// TIA Portal V17 export
// export: Created 2022-06-27T13:58:59.0889884Z, ExportSetting WithDefaults, DisplayName Totally Integrated Automation Portal, DisplayVersion V17 Update 3, DisplayName TIA Portal Openness, DisplayVersion V17 Update 3, DisplayName TIA Portal Version Control Interface, DisplayVersion V17, DisplayName SINAMICS Startdrive Advanced, DisplayVersion V17 Update1, DisplayName SINAMICS Startdrive G110M, G120, G120C, G120D, G120P, G115D, DisplayVersion V17 Update1, DisplayName SINAMICS Startdrive G130, G150, S120, S150, SINAMICS MV, S210, DisplayVersion V17 Update1, DisplayName STEP 7 Professional, DisplayVersion V17 Update 3, DisplayName STEP 7 Safety, DisplayVersion V17, DisplayName WinCC UA Professional, DisplayVersion V17 Update 3
FUNCTION_BLOCK "S063_PROTECTION"   // FB63, LAD
{ S7_Optimized_Access := 'TRUE' }
VERSION : 0.1
// stored: AutoNumber false, IsIECCheckEnabled false, IsRetainMemResEnabled false, MemoryReserve 100, SetENOAutomatically false, UDAEnableTagReadback false
BEGIN

REGION Network 1: F32-2C - Burner Fan
END_REGION

REGION Network 2: F33-4C - Roaster Cyclone Rotary Valve
END_REGION

REGION Network 3: F33-6C - Water Pump
END_REGION

REGION Network 4: F34-2C - Roaster Fan
END_REGION

REGION Network 5: F34-4C - Dryer Fan
END_REGION

REGION Network 6: F34-6C - Cooler Fan
END_REGION

REGION Network 7: F35-2C - Roasting Chamber 1
END_REGION

REGION Network 8: F35-4C - Roasting Chamber 2
END_REGION

REGION Network 9: F36-2C - Chamber 1 Ambient Air Blower
END_REGION

REGION Network 10: F36-3C - Chamber 2 Ambient Air Blower
END_REGION

REGION Network 11: F36-5C - Cooler Cyclone Rotary Valve
END_REGION

REGION Network 12: F36-7C - Cooler Conveyor Belt
END_REGION

REGION Network 13: F36-8C - Tilted Conveyor Belt
END_REGION

REGION Network 14: F37-2C - Cooler Chamber 1
END_REGION

REGION Network 15: F37-3C - Cooler Chamber 2
END_REGION

REGION Network 16: F37-5C - Rotary Valve Drying Chamber 1 Cyclone
END_REGION

REGION Network 17: F37-7C - Rotary Valve Drying Chamber 2 Cyclone
END_REGION

REGION Network 18: F37-8C - Cyclones Screw Conveyor
END_REGION
END_FUNCTION_BLOCK
